FUNCTION_BLOCK TC_InputMapping (* Service Interface Function Block Type *)
  (* Standard: ISO 11783-10; Function: All Inputs; Type: TC according to ISO 11783-10; Description: Copyright (c) 2018, 2023 Jose Cabral, HR Agrartechnik GmbH This program and the accompanying materials are made available under the terms of the Eclipse Public License 2.0 which is available at https://www.eclipse.org/legal/epl-2.0/ SPDX-License-Identifier: EPL-2.0 this maps to ID 32 bit Process Data (PD) *)
  (* Version 1.0, 2018-12-05, Jose Cabral *)
  (* Version 1.1, 2022-08-04, Franz Höpfinger, HR Agrartechnik GmbH *)
  (* Version 1.2, 2023-01-05, Franz Höpfinger, HR Agrartechnik GmbH *)
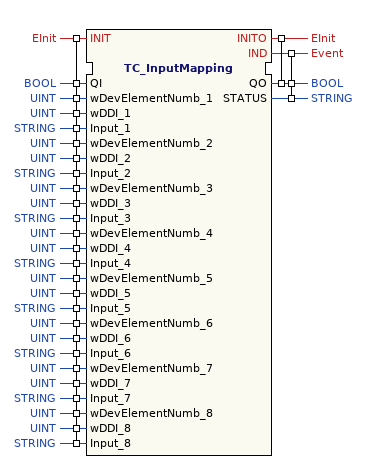
  EVENT_INPUT
    INIT : EInit WITH QI, wDevElementNumb_1, wDDI_1, Input_1, wDevElementNumb_2, wDDI_2, Input_2, wDevElementNumb_3, wDDI_3, Input_3, wDevElementNumb_4, wDDI_4, Input_4, wDevElementNumb_5, wDDI_5, Input_5, wDevElementNumb_6, wDDI_6, Input_6, wDevElementNumb_7, wDDI_7, Input_7, wDevElementNumb_8, wDDI_8, Input_8; (* Service Initialization *)
  END_EVENT
  EVENT_OUTPUT
    INITO : EInit WITH QO; (* Initialization Confirm *)
    IND WITH QO, STATUS; (* Indication from Resource *)
  END_EVENT
  VAR_INPUT
    QI : BOOL; (* Event Input Qualifier *)
    wDevElementNumb_1 : UINT; (* Requested element number of TC of Input 1 *)
    wDDI_1 : UINT; (* Data dictionary identifier of Input 1 *)
    Input_1 : STRING; (* Identifier for Input 1 *)
    wDevElementNumb_2 : UINT; (* Requested element number of TC of Input 2 *)
    wDDI_2 : UINT; (* Data dictionary identifier of Input 2 *)
    Input_2 : STRING; (* Identifier for Input 2 *)
    wDevElementNumb_3 : UINT; (* Requested element number of TC of Input 3 *)
    wDDI_3 : UINT; (* Data dictionary identifier of Input 3 *)
    Input_3 : STRING; (* Identifier for Input 3 *)
    wDevElementNumb_4 : UINT; (* Requested element number of TC of Input 4 *)
    wDDI_4 : UINT; (* Data dictionary identifier of Input 4 *)
    Input_4 : STRING; (* Identifier for Input 4 *)
    wDevElementNumb_5 : UINT; (* Requested element number of TC of Input 5 *)
    wDDI_5 : UINT; (* Data dictionary identifier of Input 5 *)
    Input_5 : STRING; (* Identifier for Input 5 *)
    wDevElementNumb_6 : UINT; (* Requested element number of TC of Input 6 *)
    wDDI_6 : UINT; (* Data dictionary identifier of Input 6 *)
    Input_6 : STRING; (* Identifier for Input 6 *)
    wDevElementNumb_7 : UINT; (* Requested element number of TC of Input 7 *)
    wDDI_7 : UINT; (* Data dictionary identifier of Input 7 *)
    Input_7 : STRING; (* Identifier for Input 7 *)
    wDevElementNumb_8 : UINT; (* Requested element number of TC of Input 8 *)
    wDDI_8 : UINT; (* Data dictionary identifier of Input 8 *)
    Input_8 : STRING; (* Identifier for Input 8 *)
  END_VAR
  VAR_OUTPUT
    QO : BOOL; (* Event Output Qualifier *)
    STATUS : STRING; (* Service Status *)
  END_VAR
END_FUNCTION_BLOCK
